# EPICS substitutions: modules/event/evrSupport/Db/ioc/IOC-IN20-LS11evr.substitutions
#==============================================================================
#
# Abs:  LCLS EVR IOC records for IN20 LS11
#
# Name: IOC-IN20-LS11evr.substitutions
#
#==============================================================================
#
file evrLSXX.db
{
pattern { DEVICE        }
	{ EVR:IN20:LS11 }
}
